FUNCTION_BLOCK FB_HE_SolidAttenuatorSettings EXTENDS FB_Fallible IMPLEMENTS I_HE_SolidAttenuatorSettings
VAR
END_VAR

{warning 'Add method implementation '}
METHOD GetError : BOOL
END_METHOD

{warning 'Add method implementation '}
METHOD GetErrorMsg : lcls_twincat_physics.T_MaxString
END_METHOD

{warning 'Add method implementation '}
METHOD GetSettings
VAR_IN_OUT
    Settings	: ST_HE_SolidAttenuatorSettings;
END_VAR
END_METHOD

END_FUNCTION_BLOCK

(* stored: Version 1.1.0.1
   POU FB_HE_SolidAttenuatorSettings: Id {b7aeb9ae-a678-4241-8eb7-e9abac20fe60}, SpecialFunc None
   Method GetError: Id {f0dcfe04-9fed-4c52-b54f-abd1e817b16e}
   Method GetErrorMsg: Id {43195afd-0baf-4c0d-9893-607711c1a374}
   Method GetSettings: Id {5f1c848b-6ca6-4711-a071-64cd22ef5930} *)
